FUNCTION_BLOCK FB_SIM_MOTOR
VAR_IN_OUT
	stSimMotor	:	DUT_SimMotor;
END_VAR
VAR_OUTPUT
	bMoving		:	BOOL := FALSE;
END_VAR
VAR
	fCurrPos	:	LREAL := stSimMotor.fPosition;
	fReqPos		:	LREAL := stSimMotor.fPosition;
	fbTimer		:	TON;
	fTravelTime	:	REAL;
	STATE		:	DUT_SimMotorStates;
	xFirstPass	:	BOOL := TRUE;
END_VAR

(* On first PLC pass, put valve into init state*)
IF xFirstPass THEN
	STATE := DUT_SimMotorStates.IDLE;
	xFirstPass := FALSE;
END_IF

fReqPos := stSimMotor.fPosition;

CASE STATE OF

	DUT_SimMotorStates.IDLE:
		bMoving := FALSE;
		IF fReqPos <> fCurrPos THEN
			STATE := DUT_SimMotorStates.CHECK;
		END_IF
		
		
	DUT_SimMotorStates.CHECK:
		IF fReqPos > fCurrPos THEN // Check OK to move forward
			IF stSimMotor.bAllEnable OR stSimMotor.bAllForwardEnable THEN
				STATE := DUT_SimMotorStates.MOVING;
			ELSE
				STATE := DUT_SimMotorStates.IDLE;
			END_IF
		ELSE IF fReqPos < fCurrPos THEN // Check OK to move backward
			IF stSimMotor.bAllEnable OR stSimMotor.bAllBackwardEnable THEN
				STATE := DUT_SimMotorStates.MOVING;
			ELSE
				STATE := DUT_SimMotorStates.IDLE;
			END_IF
		ELSE // Somthing weird happened; should never get to this state. Just go back to idle. 
			STATE := DUT_SimMotorStates.IDLE;
		END_IF
		END_IF
	
	
	DUT_SimMotorStates.MOVING:
//		IF stSimMotor.fVelocity = 0.0 THEN
//			stSimMotor.fVelocity := 1.0; // set velocity to reasonable value; prevent divide by zero
//		END_IF
//		fTravelTime := ABS((fReqPos - fCurrPos)/stSimMotor.fVelocity)
		fbTimer(PT:=T#3S, IN:=TRUE);
		bMoving := TRUE;
		
		IF fbTimer.Q = TRUE THEN // time has elapsed
			fbTimer.IN := FALSE;
			stSimMotor.fPosition := fReqPos;
			fCurrPos := fReqPos;
			STATE := DUT_SimMotorStates.IDLE;
		END_IF
END_CASE

END_FUNCTION_BLOCK

(* stored: Version 1.1.0.1, ProductVersion 3.1.4024.2
   POU FB_SIM_MOTOR: Id {8583a234-1d69-4506-be3c-a0ed673500be}, SpecialFunc None *)
